Omron Sysmac Studio project Convert (Sysmac Studio 1.65.0.64007, StandardProject)

# Controller new_Controller_0: NX1P2-1040DT1 version 1.69
Task PrimaryTask (priority 4, period or condition 2000): Program0

VAR_GLOBAL
    Trunc_Var : DINT;
    Round_Var : DINT;
    RoundUp_Var : DINT;
END_VAR

PROGRAM Program0
VAR_EXTERNAL
    Trunc_Var : DINT;
    Round_Var : DINT;
    RoundUp_Var : DINT;
END_VAR

(* Section Section0: ladder, written here as Structured Text *)

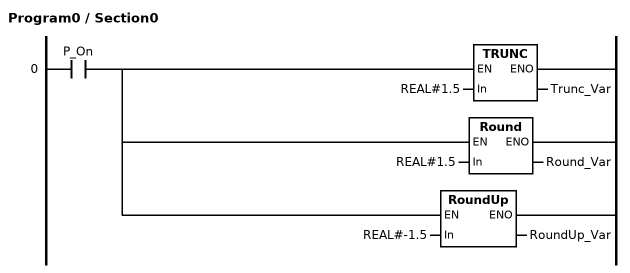
(* Rung 0 *)
IF P_On THEN
    Trunc_Var := TRUNC(In := REAL#1.5);
    Round_Var := Round(In := REAL#1.5);
    RoundUp_Var := RoundUp(In := REAL#-1.5);
END_IF;
END_PROGRAM